// TIA Portal V20 export
DATA_BLOCK "DB_Manual"   // DB4
// stored: Access Published, MemoryReserve 100, Namespace LineA1
   VAR
      Conveyor : Struct
         ID : Int;
         Enable : Bool;
         Run : Bool;
         in : Bool;
      END_STRUCT;
      Line : Struct
         A1 : Struct
            Conveyor { S7_SetPoint := 'True'} : Array[_.minA1.._.maxA1] of "LineA1.ManualInputs";
         END_STRUCT;
      END_STRUCT;
   END_VAR
BEGIN
END_DATA_BLOCK
